Staubli VAL3: CircleCenter.dtx

bool bExit
public bool bFrameSave = true
bool bFrameTeach
bool bOk = true
bool bSame = true
frame fFrame1 = {x=1612.412783, y=41.853304, z=-98.136139, rx=-0.102691, ry=-0.966077, rz=-75.481347, fatherId=world[0]}
frame fFrameRef = {fatherId=world[0]}
mdesc mNomSpeed
num nAngle = 75.485802
num nDia = 298.39416
num nFrame1Err = -1
num nItem[6]
num nMax[6]
num nMin[6]
num nSelectedPt = 2
num nStatus = 6
num nWorkingMode = 1
public pointRx pFrameRefPt[3]
  [0] = {x=1649.443256, y=-101.6459, z=-97.721003, rx=0.130916, ry=-179.947483, rz=21.208766, shoulder=lefty, elbow=epositive, wrist=wpositive, fatherId=world[0]}
  [1] = {x=1756.967626, y=82.83778, z=-95.770129, rx=0.131083, ry=-179.947766, rz=21.208255, shoulder=lefty, elbow=epositive, wrist=wpositive, fatherId=world[0]}
  [2] = {x=1467.188622, y=8.3784, z=-100.569453, rx=0.130753, ry=-179.947125, rz=21.208996, shoulder=lefty, elbow=epositive, wrist=wpositive, fatherId=world[0]}
pointRx pPointCenter = {x=1612.412783, y=41.853304, z=-98.136139, rx=-0.102691, ry=-0.966077, rz=60.039915, fatherId=world[0]}
string sButton[2]
  [0] = "是"
  [1] = "否"
string sCutPosStatus
string sEmptyOrNotC[3]
string sItem[6]
string sOffSet[6]
  [0] = "X:  1612.41"
  [1] = "Y:  41.85"
  [2] = "Z:  -98.14"
  [3] = "Rx: -0.1 "
  [4] = "Ry: -0.97"
  [5] = "Rz: -75.48"
string sThreeOffset[3]
  [0] = "第1点(圆周上)"
  [1] = "第2点(圆周上)"
  [2] = "第3点(圆周上)"
tool tTool = {x=350.22, y=-0.767094, z=232.538993, rx=-89.841339, ry=89.729222, rz=89.842087, fatherId=flange[0], ioLink=valve1}
trsf trFrame
trsf trOffSetOut
trsf trOffset = {x=1612.412783, y=41.853304, z=-98.136139, rx=-0.102691, ry=-0.966077, rz=-75.481347}
